KUKA KRL program: ZAMKN_CHWYTAK.src

&ACCESS RVP
&REL 9
&PARAM TEMPLATE = C:\KRC\Roboter\Template\ExpertVorgabe
&PARAM EDITMASK = *
DEF ZAMKN_CHWYTAK( )

PULSE($OUT[5],TRUE,3)
PULSE($OUT[6],TRUE,3)
WAIT FOR $OUT[6] == FALSE

END
